FUNCTION_BLOCK FB_FallibleMock IMPLEMENTS I_Fallible
VAR
    bError : BOOL;
    sErrorMsg : T_MaxString;
END_VAR


METHOD ClearError

bError := FALSE;
sErrorMsg := '';
END_METHOD


METHOD GetError : BOOL

GetError := bError;
END_METHOD


METHOD GetErrorMsg : T_MaxString

GetErrorMsg := sErrorMsg;
END_METHOD


METHOD PUBLIC SetError
VAR_INPUT
    sMsg : T_MaxString;
END_VAR

bError := TRUE;
sErrorMsg := sErrorMsg;
END_METHOD

END_FUNCTION_BLOCK

(* stored: Version 1.1.0.1
   POU FB_FallibleMock: Id {cb18ced6-2ac4-4212-bee1-29e44a52e6ff}, SpecialFunc None
   Method ClearError: Id {2ddf41ad-3436-4862-aa14-18fd1b132b45}
   Method GetError: Id {5ab80806-3fc1-498b-86c4-0101756110fd}
   Method GetErrorMsg: Id {e03e4837-0e6a-440b-875b-fd2f0dfdd389}
   Method SetError: Id {a477b405-4fe1-4496-8d2b-156cca50a0de} *)
